(* PLC project Unnamed, Unknown Unnamed 1 *)
(* stored: creationDateTime 2026-08-06T10:18:11, modificationDateTime 2026-08-06T10:18:11 *)

PROGRAM main
  VAR
    Wind_Speed AT %QW0 : INT;  (* Menerima data kecepatan angin dari Node-RED *)
    Wind_Dir AT %QW1 : INT;  (* Menerima sudut arah angin dari Node-RED *)
    Runway_Head AT %QW2 : INT;  (* Sudut arah landasan pacu (bisa diatur dari Node-RED) *)
    Crosswind_Val AT %MD10 : REAL;  (* Variabel internal untuk menyimpan hasil hitung matematika *)
    Alarm_Aman AT %QX0.0 : BOOL;  (* Output logika untuk status aman (Hijau) *)
    Alarm_Waspada AT %QX0.1 : BOOL;  (* Output logika untuk status waspada (Kuning) *)
    Alarm_Bahaya AT %QX0.2 : BOOL;  (* Output logika untuk status bahaya (Merah) *)
  END_VAR
  VAR
    Selisih_Sudut : INT;  (* Menyimpan hasil pengurangan (SUB) antara arah angin dan arah landasan pacu. Hasilnya masih berupa bilangan bulat (Derajat). *)
    Sudut_Real : REAL;  (* Menyimpan nilai Selisih_Sudut yang sudah diubah formatnya menjadi desimal menggunakan blok INT_TO_REAL. *)
    Cek_Aman : BOOL;
    Cek_Waspada : BOOL;
    Cek_Bahaya : BOOL;
    Hasil_GE : BOOL;
    Hasil_LT : BOOL;
    Sudut_Radian : REAL;  (* Menyimpan hasil perkalian Sudut_Real dengan konstanta 0.0174533. Konversi dari Derajat ke Radian ini wajib dilakukan karena blok SIN di PLC hanya membaca satuan Radian. *)
    Kecepatan_Real : REAL;  (* Menyimpan data kecepatan angin awal yang diubah formatnya menjadi desimal (dengan INT_TO_REAL) agar bisa dikalikan dengan bilangan desimal lainnya. *)
    Nilai_Sinus : REAL;  (* Menyimpan nilai sinus yang dihasilkan dari blok matematika SIN. *)
    Hasil_SUB : INT;
    Hasil_MUL : INT;
    Val_Radian : REAL := 0.0174533;
    Batas_Aman : REAL := 15.0;
    Batas_Bahaya : REAL := 25.0;
  END_VAR

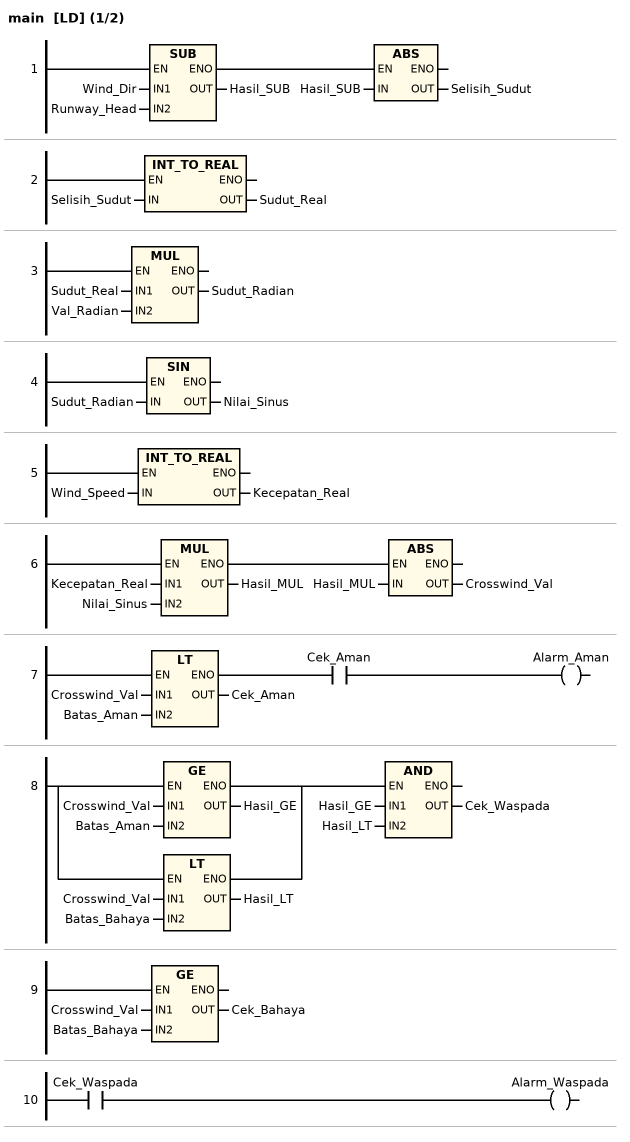
(* LD diagram, written out as Structured Text *)
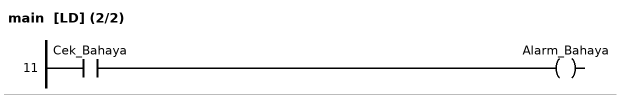
Alarm_Aman := Cek_Aman;
Alarm_Waspada := Cek_Waspada;
Alarm_Bahaya := Cek_Bahaya;
Hasil_SUB := Wind_Dir - Runway_Head;
Selisih_Sudut := ABS(Hasil_SUB);
Sudut_Real := INT_TO_REAL(Selisih_Sudut);
Sudut_Radian := Sudut_Real * Val_Radian;
Nilai_Sinus := SIN(Sudut_Radian);
Kecepatan_Real := INT_TO_REAL(Wind_Speed);
Hasil_MUL := Kecepatan_Real * Nilai_Sinus;
Crosswind_Val := ABS(Hasil_MUL);
Cek_Aman := Crosswind_Val < Batas_Aman;
Hasil_GE := Crosswind_Val >= Batas_Aman;
Hasil_LT := Crosswind_Val < Batas_Bahaya;
Cek_Waspada := Hasil_GE AND Hasil_LT;
Cek_Bahaya := Crosswind_Val >= Batas_Bahaya;
END_PROGRAM

CONFIGURATION Config0
  RESOURCE Res0 ON PLC
    TASK task0(INTERVAL := T#20ms, PRIORITY := 1);
    PROGRAM instance0 WITH task0 : main;
  END_RESOURCE
END_CONFIGURATION
